{attribute addProperty BoxType "EL3413-0000-0016"}
{attribute addProperty Id "IndexAT %Q*USINT811ChannelAT %Q*USINT812"}
{attribute addProperty CRC "1097446643"}
{attribute addProperty SizeInBites "16"}
{attribute addProperty SizeInBytes "2"}
TYPE PM_Outputs_Auxiliary_4169B4F3 :
STRUCT
	{attribute addProperty Name "Index"}
	Index AT %Q* : USINT;
	{attribute addProperty Name "Channel"}
	Channel AT %Q* : USINT;
END_STRUCT
END_TYPE

(* stored: Version 1.2.0.0, ProductVersion 3.1.4024.9
   DUT PM_Outputs_Auxiliary_4169B4F3: Id {6365831f-5200-4508-b368-15991f5999de} *)
